FUNCTION f_to_Period : REAL
VAR_INPUT
	fFrequency : REAL;
END_VAR
VAR	
	fFracOfTime			: REAL;
	fReferenceTimeTemp	: REAL;	
END_VAR

IF fFrequency <> 0 THEN
	fFracOfTime	:= (1/fFrequency);
END_IF

fReferenceTimeTemp	:= TIME_TO_REAL(T#1MS);

f_to_Period	:= fReferenceTimeTemp * fFracOfTime;

END_FUNCTION

(* stored: Version 1.1.0.1, ProductVersion 3.1.4024.6
   POU f_to_Period: Id {e957decd-057e-401d-ad93-1f9d94d5157e}, SpecialFunc None *)
